(* CODESYS project veibom.export

Project tree, tasks and I/O mapping:
  Device : CODESYS Control Win V3, 3S - Smart Software Solutions GmbH, version 3.5.16.30
    application Application
      libraries: Standard, * (System)
      task MainTask (cyclic, interval t#20ms, priority 1) calls PLC_PRG
      task VISU_TASK (cyclic, interval 100 ms, priority 31) calls VisuElems.Visu_Prg
      program PLC_PRG [CFC]
      function block Veibom [ST]
      visualisation Visualization
*)

// Device/Application/PLC_PRG
PROGRAM PLC_PRG
VAR
	mekanisme: veibom;
	vektplate: BOOL;
	fjernkotroll: BOOL;
	Mek: Veibom;
END_VAR

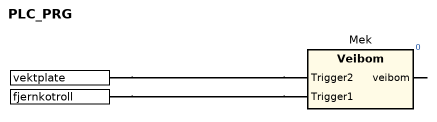
Mek(Trigger2 := vektplate, Trigger1 := fjernkotroll); // Veibom

END_PROGRAM

// Device/Application/Veibom
FUNCTION_BLOCK Veibom
VAR_INPUT
	Trigger1 : BOOL;
	trigger2: BOOL;
END_VAR
VAR_OUTPUT
	veibom : BOOL;
END_VAR
VAR
END_VAR

IF Trigger1 = TRUE AND trigger2 = TRUE THEN
	Veibom := TRUE;
END_IF

IF Trigger1 = FALSE AND trigger2 = TRUE THEN
	Veibom := FALSE;
END_IF

IF Trigger1 = TRUE AND trigger2 = FALSE THEN
	Veibom := FALSE;
END_IF

IF Trigger1 = FALSE AND trigger2 = FALSE THEN
	Veibom := FALSE;
END_IF

END_FUNCTION_BLOCK

// Device/Application/Visualization
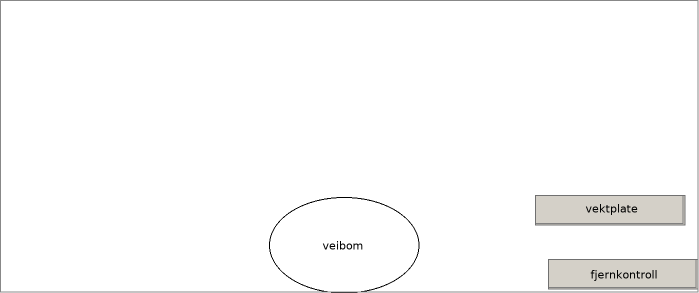
VISUALIZATION Visualization  // 699x293
    Button (535,195 150x30)
        toggle PLC_PRG.vektplate
    Button (548,259 150x30)
        toggle PLC_PRG.fjernkotroll
    Ellipse (269,197 150x96)
        toggle PLC_PRG.Mek.veibom
    Label (537,194 150x30), "vektplate"
    Label (549,260 150x30), "fjernkontroll"
    Label (268,231 150x30), "veibom"
END_VISUALIZATION
